FUNCTION_BLOCK JUnitResultFile
VAR_GENERIC CONSTANT
	_MaxTestSuiteCount : DINT := 10;
END_VAR IMPLEMENTS I_UnitTestResultFile
VAR
	_Initialized, Write										   : BOOL;
	XmlDomParser											   : FB_XmlDomParser;
	RootNode, TestSuitesNode, TestSuite, TestCase, TestCaseSub : SXmlNode;
	_Path													   : STRING;
	SuiteNames												   : ARRAY[0.._MaxTestSuiteCount] OF STRING;
	SuiteNodes												   : ARRAY[0.._MaxTestSuiteCount] OF SXmlNode;
	SuiteCount												   : DINT;
	DoneMessage												   : FB_TcMessage;
	Source													   : FB_TcSourceInfo;
	_SuiteOverflowCount										   : UDINT;
END_VAR

METHOD AddTestCaseResult
VAR_INPUT
	TestClassName	: STRING;
	TestName		: STRING;
	Duration		: LREAL;
	FailureMessage : STRING := '';
	FailureType	: STRING := '';
	FailureNote	: STRING := '';
END_VAR
VAR
	SuiteNode : SXmlNode;
END_VAR
IF NOT Initialized THEN
	RETURN;
END_IF

SuiteNode := FindSuiteNode(TestClassName);
IF SuiteNode = 0 THEN
	RETURN;
END_IF

TestCase := XmlDomParser.AppendChild(SuiteNode,
									 'testcase',
									 '',
									 FALSE);

XmlDomParser.AppendAttribute(TestCase, 'classname', TestClassName);
XmlDomParser.AppendAttribute(TestCase, 'name', TestName);
XmlDomParser.AppendAttributeAsDouble(TestCase, 'time', Duration);
IF FailureType <> '' THEN
	TestCaseSub := XmlDomParser.AppendChild(TestCase,
											'failure',
											FailureNote,
											FALSE);

	XmlDomParser.AppendAttribute(TestCaseSub, 'message', FailureMessage);
	XmlDomParser.AppendAttribute(TestCaseSub, 'type', FailureType);
END_IF
END_METHOD

METHOD AddTestSuite
VAR_INPUT
	Name : STRING;
END_VAR
VAR
	ResultString : T_MaxString;
END_VAR
IF NOT Initialized THEN
	RETURN;
END_IF

// Reuse the existing node if this suite name was already added (shared result file across multiple TestSuite instances)
TestSuite := FindSuiteNode(Name);
IF TestSuite <> 0 THEN
	RETURN;
END_IF

TestSuite := XmlDomParser.AppendChild(TestSuitesNode,
									  'testsuite',
									  '',
									  FALSE);

XmlDomParser.AppendAttribute(TestSuite, 'name', name);

IF SuiteCount <= _MaxTestSuiteCount THEN
	SuiteNames[SuiteCount] := Name;
	SuiteNodes[SuiteCount] := TestSuite;
	SuiteCount			   := SuiteCount + 1;
ELSE
	_SuiteOverflowCount := _SuiteOverflowCount + 1;

	Source.sName := Name;
	DoneMessage.Create(eventClass	:= TC_EVENT_CLASSES.TestEvents,
					   nEventId		:= 1,
					   eSeverity	:= TcEventSeverity.Error,
					   ipSourceInfo := Source);

	ResultString := CONCAT('TestSuite not added, max TestSuites exeeded - ', TO_STRING(_MaxTestSuiteCount));
	DoneMessage.ipArguments.AddString(ResultString);
	DoneMessage.Send(0);
	Source.Clear();
	DoneMessage.Release();
END_IF
END_METHOD

METHOD AddTestSuiteStatistics
VAR_INPUT
	Name	  : STRING;
	Tests	  : UDINT;
	Failures : UDINT := 0;
	Errors	  : UDINT := 0;
	Skipped	  : UDINT := 0;
	Duration  : LREAL;
END_VAR
VAR
	SuiteNode : SXmlNode;
END_VAR
IF NOT Initialized THEN
	RETURN;
END_IF

SuiteNode := FindSuiteNode(Name);
IF SuiteNode = 0 THEN
	RETURN;
END_IF

XmlDomParser.AppendAttributeAsUint(SuiteNode, 'tests', Tests);
XmlDomParser.AppendAttributeAsUint(SuiteNode, 'failures', Failures);
XmlDomParser.AppendAttributeAsUint(SuiteNode, 'errors', Errors);
XmlDomParser.AppendAttributeAsUint(SuiteNode, 'skipped', Skipped);
XmlDomParser.AppendAttributeAsDouble(SuiteNode, 'time', Duration);
END_METHOD

METHOD Cyclic
XmlDomParser.SaveDocumentToFile(_Path, Write);
END_METHOD

//FB_Init is always available implicitly and it is used primarily for initialization.

//The return value is not evaluated. For a specific influence, you can also declare the

//methods explicitly and provide additional code there with the standard initialization

//code. You can evaluate the return value.
METHOD FB_Init : BOOL
VAR_INPUT
	bInitRetains : BOOL; // TRUE: the retain variables are initialized (reset warm / reset cold)
	bInCopyCode	 : BOOL; // TRUE: the instance will be copied to the copy code afterward (online change)
	Path		 : STRING;
END_VAR
_Path := Path;
END_METHOD

METHOD PRIVATE FindSuiteNode : SXmlNode
VAR_INPUT
	Name : STRING;
END_VAR
VAR
	i : DINT;
END_VAR
FindSuiteNode := 0;

FOR i := 0 TO SuiteCount - 1 DO
	IF SuiteNames[i] = Name THEN
		FindSuiteNode := SuiteNodes[i];
		RETURN;
	END_IF
END_FOR
END_METHOD

METHOD Initialize
VAR_INPUT
	ReInitialize : BOOL := FALSE;
END_VAR
IF Initialized AND NOT ReInitialize THEN
	RETURN;
END_IF

XmlDomParser.NewDocument();
RootNode	   := XmlDomParser.GetDocumentNode();
TestSuitesNode := XmlDomParser.AppendChild(RootNode,
										   'testsuites',
										   '',
										   FALSE);

SuiteCount	 := 0;
_Initialized := TRUE;
END_METHOD

{attribute 'monitoring' := 'call'}
PROPERTY Initialized : BOOL
GET
Initialized := _Initialized;
END_GET
END_PROPERTY

{attribute 'monitoring' := 'call'}
PROPERTY Path : STRING
SET
_Path := Path;
END_SET
END_PROPERTY

METHOD SaveResult
IF NOT Initialized THEN
	RETURN;
END_IF

Write := TRUE;
END_METHOD

{attribute 'monitoring' := 'call'}
PROPERTY SuiteOverflowCount : UDINT
GET
SuiteOverflowCount := _SuiteOverflowCount;
END_GET
END_PROPERTY

END_FUNCTION_BLOCK

(* stored: Version 1.1.0.1
   POU JUnitResultFile: Id {467a2f7d-ea77-463d-bccb-4ff68e52df26}, SpecialFunc None
   Method AddTestCaseResult: Id {fef2152d-9883-418e-81df-19425d45758e}
   Method AddTestSuite: Id {b9ed6143-3d62-40dc-ab57-7f199b7a8267}
   Method AddTestSuiteStatistics: Id {37965891-a54c-4d6f-81af-5996d77b7537}
   Method Cyclic: Id {4a8e3fe5-235e-4dba-86c7-512836695edb}
   Method FB_Init: Id {5f9e5f1d-2f0b-4d1a-8a7e-9c3a1e6b4d2f}
   Method FindSuiteNode: Id {8c1f2e3d-4b5a-4c6d-9e7f-0a1b2c3d4e5f}
   Method Initialize: Id {23d2b239-3906-4cef-b04c-0fd9ab13f256}
   Property Initialized: Id {3d7d628e-0047-482f-96af-148144f8b22c}
   Get Get: Id {998aca69-b6fa-4c38-a66e-64b2cd84ac9d}
   Property Path: Id {61e6a68d-66c6-4093-b352-4efc4872d68b}
   Set Set: Id {4e012c2e-dd46-405f-b43e-4e46079d4b27}
   Method SaveResult: Id {24be214b-5fc2-42d3-8a34-ff3a2fc199dd}
   Property SuiteOverflowCount: Id {2b3c4d5e-6f70-4a81-9b2c-3d4e5f607182}
   Get Get: Id {3c4d5e6f-7081-4a92-8b3c-4d5e60718293} *)
